(* IEC 61131-3 sources: SHU_NSTV/CodeSys_Project, 5 files *)

(* ---- Struct_BY.st ---- *)
TYPE Struct_BY :
STRUCT
	// Команды
	//xOpen, xClose, xStop, xReset : BOOL;
	Auto_xOpen, Auto_xClose, Auto_xStop, Auto_xReset : BOOL;
	Service_xOpen, Service_xClose, Service_xStop, Service_xReset : BOOL;
	ConditionToxOpen, ConditionToxClose, ConditionToxStop, ConditionToxAutoStop, ConditionToxReset : BOOL;
	sOpen, sClose, sStop, sReset : FB_SignalSplit;
	rtrig_xOpen, rtrig_xClose, rtrig_xStop, rtrig_xReset : R_TRIG;
	autoCmdWord : Union_ByteToWord;
	// Статусы
	xStatusOpen, xStatusClosed, xStatusStopped, xStatusError, xStatusReady, xStatusKmOpen, xStatusKmClose : BOOL;
	xOpenProcess, xCloseProcess : BOOL;
	StatusShutter : INT;
	StatusMotor : INT;
	StatusRemote : INT; // 0 - Выключен, 1 - Местный, 2 - Авто
	wStatus : Union_ByteToWord;
	// Обработка ошибок
	ErrorOpen, ErrorClose, ErrorStop : Error_SignalLongExpectation;
	xLongExpectationOpen, xErrorLongExpectationClose, xErrorLongExpectationStop : BOOL;
	// Класс ЗРА
	Device : Shutter;
END_STRUCT
END_TYPE

(* ---- Struct_PU.st ---- *)
TYPE Struct_PU :
STRUCT
	// --- Команды ---
	Auto_xStartBP, Auto_xStartVFD, Auto_xStop, Auto_xSwitchToBP, Auto_xSwitchToVFD, Auto_xReset, Auto_xEmergencyStop : BOOL;
	Auto_xEnableLocalRemote : BOOL; // Разрешение на местное управление насосом
	Auto_xRequestLocalRemote : BOOL; // Запрос на местное управление

	Auto_cmdWord : Union_ByteToWord;
	Auto_cmdSetFreqWord : Union_RealToWord;

	Service_xStartBP, Service_xStartVFD, Service_xStop, Service_xSwitchToBP, Service_xSwitchToVFD, Service_xReset, Service_xEmergencyStop : BOOL;
	xConditionToStartBP, xConditionToStartVFD, xConditionToSwitchToBP, xConditionToSwitchToVFD, xConditionToStop, xConditionToAutoStop : BOOL; // Условия выполнения команд

	rtrig_xStartBP        : R_TRIG;
	rtrig_xStartVFD       : R_TRIG;
	rtrig_xStop           : R_TRIG;
	rtrig_xSwitchToBP     : R_TRIG;
	rtrig_xSwitchToVFD    : R_TRIG;
	rtrig_xReset          : R_TRIG;
	rtrig_xEmergencyStop  : R_TRIG;

	ErrorxStartBP         : Error_SignalLongExpectation;
	ErrorxStartVFD        : Error_SignalLongExpectation;
	ErrorxStop            : Error_SignalLongExpectation;
	ErrorxSwitchToBP      : Error_SignalLongExpectation;
	ErrorxSwitchToVFD     : Error_SignalLongExpectation;

	// --- Состояния ---
	// Дискретные входы
	xStatusEnableBP       : BOOL;
	xStatusEnableVFD      : BOOL;
	xStatusManual         : BOOL;
	xManualStart          : BOOL;
	xManualStop           : BOOL;
	xStatusDry            : BOOL;
	// Генерируемые состояния
	xCommonError          : BOOL;
	xEmergencyStopStatus  : BOOL;

	xErrorLongTimeException_xStartBP     : BOOL;
	xErrorLongTimeException_xStartVFD    : BOOL;
	xErrorLongTimeException_xStop        : BOOL;
	xErrorLongTimeException_xSwitchToBP  : BOOL;
	xErrorLongTimeException_xSwitchToVFD : BOOL;

	xErrorLostFeedbackSignal  : BOOL;
	xErrorEnableStatusVFD : BOOL;

	xReadyToStartBP       : BOOL;
	xReadyToStartVFD      : BOOL;

	iStatus               	: INT;
	wStatus					: Union_ByteToWord;
	wCurrentSpeed			: Union_RealToWord;

	ton_ErrorLostFeedbackSignal : TON;

	// --- Класс насоса ---
	Device : Pump_VFD;

	// --- Предпусковая сигнализация ---
	cmdStartBP_StartSound      	: FB_StartSiren;
	cmdStartVFD_StartSound		: FB_StartSiren;
	xSoundSirenSetSound  : BOOL;
END_STRUCT

END_TYPE

(* ---- Struct_VFD.st ---- *)
TYPE Struct_VFD :
STRUCT
	// Команды
	//xStart, xStop, xEmergencyStop, xReset, xSetToMain, xSetToReserve : BOOL;
	Auto_Start, Auto_Stop, Auto_EmergencyStop, Auto_Reset, Auto_SetToMain, Auto_SetToReserve : BOOL;
	Service_Start, Service_Stop, Service_EmergencyStop, Service_Reset, Service_SetToMain, Service_SetToReserve : BOOL;
	ConditionStart, ConditionStop, ConditionEmergencyStop, ConditionReset, ConditionSetToMain, ConditionSetToReserve, ConditionAutoStop : BOOL;
	rtrig_xStart, rtrig_xStop, rtrig_xEmergencyStop, rtrig_xReset, rtrig_xSetToMain, rtrig_xSetToReserve : R_TRIG;
	// Статусы
	xPower, xFailure, xWork, xManual, xReady 	: BOOL;
	xVariableWork : BOOL; // Для проверки совпадения с переменной фактической работы
	irFrequency : REAL; // Значение частоты в Гц от модуля аналогового входа
	qrFrequency : REAL; // Значение частоты в Гц от класса
	qiScaledFrequency_0_1000 : UINT; // Значение частоты от 0 до 1000 для задачи в модуль аналогового выхода

	// --- Передача состояний по птороколу Modbus ---
	// Аналоговый выход
	wStatusOutFrequency 		: Union_RealToWord; // Выходная частота
	wStatusOutFrequencyState 	: Union_ByteToWord; // Слово состояние
	// ЧРП
	wStatusSetFrequency : Union_RealToWord; // Заданная команда
	wStatusStateCmd		: Union_ByteToWord; // Заданная команда
	wStatusState		: Union_ByteToWord; // Слово состояния
	wStatusStateError1	: Union_ByteToWord; // Слово неисправности
	wStatusUpFreqLimit	: Union_RealToWord; // Верхний предел частоты
	wStatusStateError2	: Union_ByteToWord; // Слово неисправности 2
	wStatusTorque 		: Union_RealToWord; // Значение крутящего момнета
	wStatusAO			: Union_RealToWord; // Значение АО
	// Класс ЧРП
	Device : Basic_VFD;	// Класс: базовый
END_STRUCT
END_TYPE

(* ---- Union_RealToWord.st ---- *)
TYPE Union_RealToWord :
UNION
	wTag: ARRAY [0..1] OF WORD;
	rTag: REAL;
END_UNION
END_TYPE

(* ---- FB_StartSiren.st ---- *)
FUNCTION_BLOCK FB_StartSiren
VAR_INPUT
	ixEnableSignal : BOOL; 			// Сигнал на запуск
	itFirstSoundTime : TIME;		// Время работы первого звукового сигнала
	itPauseSoundTime : TIME;		// Время работы первого звукового сигнала
	itSecondSoundTime : TIME;		// Время работы первого звукового сигнала
END_VAR
VAR_OUTPUT
	qxSound : BOOL;			// Выходной сигнал на подачу звука
	qxEndSignal : BOOL;		// Выходной сигнал об окончании работы ФБ
END_VAR
VAR
	step : INT := 0;
	xProcess : BOOL;
	ton_soundProcess : TON;
END_VAR

IF ixEnableSignal THEN
	xProcess := TRUE;
	step := 1;
END_IF;

CASE step OF
	1:
		ton_soundProcess.PT := itFirstSoundTime;
		qxSound := TRUE;
		IF ton_soundProcess.Q THEN xProcess := FALSE; step := 2; END_IF;
	2:
		qxSound := FALSE;
		ton_soundProcess.PT := itPauseSoundTime;
		xProcess := TRUE;
		IF ton_soundProcess.Q THEN xProcess := FALSE; step := 3; END_IF;
	3:
		qxSound := TRUE;
		ton_soundProcess.PT := itSecondSoundTime;
		xProcess := TRUE;
		IF ton_soundProcess.Q THEN
			xProcess := FALSE;
			qxSound := FALSE;
			step := 0;
		END_IF;
END_CASE;
ton_soundProcess(IN:= xProcess);
qxEndSignal := ton_soundProcess.Q AND step = 3;
